// TIA Portal project "Event Logger Example" (V15.1)

(* hardware
DEVICE "S71500/ET200MP station_1"  S7-1500 station
   slot 0: "Rail_0"  Rack  6ES7 590-1***0-0AA0
   slot 1: "Event Example"  CPU 1511-1 PN  6ES7 511-1AK00-0AB0  V1.8
      slot 3: "CPU display_1"  6ES7591-1AA00-0AA0
*)

// ===== PLC "Event Example"  CPU 1511-1 PN =====

VAR_GLOBAL   // PLC tag table "Default tag table"
   "System_Byte" AT %MB1 : Byte;
   "FirstScan" AT %M1.0 : Bool;
   "DiagStatusUpdate" AT %M1.1 : Bool;
   "AlwaysTRUE" AT %M1.2 : Bool;
   "AlwaysFALSE" AT %M1.3 : Bool;
   "Clock_Byte" AT %MB0 : Byte;
   "Clock_10Hz" AT %M0.0 : Bool;
   "Clock_5Hz" AT %M0.1 : Bool;
   "Clock_2.5Hz" AT %M0.2 : Bool;
   "Clock_2Hz" AT %M0.3 : Bool;
   "Clock_1.25Hz" AT %M0.4 : Bool;
   "Clock_1Hz" AT %M0.5 : Bool;
   "Clock_0.625Hz" AT %M0.6 : Bool;
   "Clock_0.5Hz" AT %M0.7 : Bool;
   "mSendKeepAlive" AT %M2.0 : Bool;
END_VAR

TYPE "EventDataToPC"
   STRUCT
      EventCode : DInt;
      Par1 : DInt;
      Par2 : DInt;
      Par3 : DInt;
      Par4 : DInt;
      Par5 : DInt;
      Par6 : DInt;
      Par7 : DInt;
      Par8 : DInt;
   END_STRUCT;
END_TYPE

TYPE "KeepAliveToPC"
   STRUCT
      MessageType : DInt := 12;
      Flags : DInt := 1;
   END_STRUCT;
END_TYPE

DATA_BLOCK "event_IDB"   // DB12
{ S7_Optimized_Access := 'TRUE' }
VERSION : 0.1
// stored: InstanceOfName ET_GeneralEventToBuffer
"ET_GeneralEventToBuffer"
BEGIN
END_DATA_BLOCK

// folder: System blocks/Program resources

DATA_BLOCK "PCComms_ConnectDly"   // DB1
{ S7_Optimized_Access := 'TRUE' }
AUTHOR : Simatic
FAMILY : IEC
NAME : IEC_TMR
VERSION : 1.0
// stored: InstanceOfName IEC_TIMER
"IEC_TIMER"
BEGIN
END_DATA_BLOCK

DATA_BLOCK "PCComms_SendRequestTimeout"   // DB6
{ S7_Optimized_Access := 'TRUE' }
AUTHOR : Simatic
FAMILY : IEC
NAME : IEC_TMR
VERSION : 1.0
// stored: InstanceOfName IEC_TIMER
"IEC_TIMER"
BEGIN
END_DATA_BLOCK

DATA_BLOCK "tKeepAlive"   // DB8
{ S7_Optimized_Access := 'TRUE' }
AUTHOR : Simatic
FAMILY : IEC
NAME : IEC_TMR
VERSION : 1.0
// stored: InstanceOfName IEC_TIMER
"IEC_TIMER"
BEGIN
END_DATA_BLOCK

DATA_BLOCK "PCComms_DisconnectDly"   // DB9
{ S7_Optimized_Access := 'TRUE' }
AUTHOR : Simatic
FAMILY : IEC
NAME : IEC_TMR
VERSION : 1.0
// stored: InstanceOfName IEC_TIMER
"IEC_TIMER"
BEGIN
END_DATA_BLOCK

DATA_BLOCK "PCComms_ReconnectDly"   // DB11
{ S7_Optimized_Access := 'TRUE' }
AUTHOR : Simatic
FAMILY : IEC
NAME : IEC_TMR
VERSION : 1.0
// stored: InstanceOfName IEC_TIMER
"IEC_TIMER"
BEGIN
END_DATA_BLOCK

DATA_BLOCK "tEventCycler"   // DB13
{ S7_Optimized_Access := 'TRUE' }
AUTHOR : Simatic
FAMILY : IEC
NAME : IEC_TMR
VERSION : 1.0
// stored: InstanceOfName IEC_TIMER
"IEC_TIMER"
BEGIN
END_DATA_BLOCK

// folder: _EventTracking

DATA_BLOCK "PCComms_Data"   // DB300
{ S7_Optimized_Access := 'FALSE' }
VERSION : 0.1
   VAR
      CON : Struct
         RequestConnection : Bool;
         RequestReconnection : Bool;
         ErrorStatus : Word;
         ManualConnect : Bool;
         ConnectRequestONS : Bool;
         ReconnectRequestONS : Bool;
         KeepAliveONS : Bool;
      END_STRUCT;
      DIAG : Struct
         ErrorStatus : Word;
         Request : Bool;
         Result : TDiag_Status;
         NumberOfSuccesses : Int := 0;
         State : Struct
            NoConnectionData : Bool;
            ConnectionTerminated : Bool;
            EstablishingConnection : Bool;
            WaitingForConnection : Bool;
            ConnectionEstablished : Bool;
            ConnectionBeingTerminated : Bool;
            UnknownState : Bool;
            HMIState : Int;
         END_STRUCT;
      END_STRUCT;
      DISCON : Struct
         ErrorStatus : Word;
         DisconnectRequest : Bool;
         ReconnectRequest : Bool;
      END_STRUCT;
      TX : Struct
         NumberOfSuccesfulSends : Int;
         HeadPointer : Int;
         TailPointer : Int;
         MaxPointer : Int := 9;
         SendRequest : Bool;
         ManualTestWithDummyData : Bool;
         DataLengthIn : UDInt;
         DataIn : Struct
            DataLength : DInt;
            Data : Array[0..1023] of Byte;
         END_STRUCT;
         DataOut : Struct
            DataLength : DInt;
            Data : Array[0..1023] of Byte;
         END_STRUCT;
         DataBuffer : Array[0..9] of Struct
            DataLength : DInt;
            Data : Array[0..1023] of Byte;
         END_STRUCT;
         StatusSaved : Word;
      END_STRUCT;
      RX : Struct
         BytesReceived : Int;
         StatusSaved : Word;
         Data : Array[0..254] of Byte;
         NumberOfSuccesfulReceives : Int;
      END_STRUCT;
      EventDataToPC : "EventDataToPC";
      KeepAliveToPC : "KeepAliveToPC";
      Alarms : Array[0..31] of Bool;
   END_VAR
BEGIN
   Alarms[0] := FALSE;
   Alarms[1] := FALSE;
   Alarms[2] := FALSE;
   Alarms[3] := FALSE;
   Alarms[4] := FALSE;
   Alarms[5] := FALSE;
   Alarms[6] := FALSE;
   Alarms[7] := FALSE;
   Alarms[8] := FALSE;
   Alarms[9] := FALSE;
   Alarms[10] := FALSE;
   Alarms[11] := FALSE;
   Alarms[12] := FALSE;
   Alarms[13] := FALSE;
   Alarms[14] := FALSE;
   Alarms[15] := FALSE;
   Alarms[16] := FALSE;
   Alarms[17] := FALSE;
   Alarms[18] := FALSE;
   Alarms[19] := FALSE;
   Alarms[20] := FALSE;
   Alarms[21] := FALSE;
   Alarms[22] := FALSE;
   Alarms[23] := FALSE;
   Alarms[24] := FALSE;
   Alarms[25] := FALSE;
   Alarms[26] := FALSE;
   Alarms[27] := FALSE;
   Alarms[28] := FALSE;
   Alarms[29] := FALSE;
   Alarms[30] := FALSE;
   Alarms[31] := FALSE;
END_DATA_BLOCK

DATA_BLOCK "ET_TxBuffer"   // DB306
{ S7_Optimized_Access := 'TRUE' }
VERSION : 0.1
   VAR
      NextAddPoint : Int;
      LastSendPoint : Int;
      SendEvtDataToPCReq : Bool;
      Buffer : Array[1..10] of "EventDataToPC";
   END_VAR
BEGIN
END_DATA_BLOCK

DATA_BLOCK "ET_Alarms"   // DB552
{ S7_Optimized_Access := 'FALSE' }
VERSION : 0.1
   VAR
      EventCommsFlt : Bool;
   END_VAR
BEGIN
END_DATA_BLOCK

DATA_BLOCK "PCComms_Connection_DB"   // DB555
{ S7_Optimized_Access := 'TRUE' }
AUTHOR : SIMATIC
FAMILY : MC7Plus
NAME : TC_IP_v4
VERSION : 1.0
// stored: InstanceOfName TCON_IP_v4
"TCON_IP_v4"
BEGIN
   ID := 2;
   InterfaceId := 64;
   LocalPort := 2000;
   RemotePort := 10200;
   RemoteAddress.ADDR[1] := 192;
   RemoteAddress.ADDR[2] := 168;
   RemoteAddress.ADDR[3] := 100;
   RemoteAddress.ADDR[4] := 253;
END_DATA_BLOCK

DATA_BLOCK "ET_GeneralData"   // DB700
{ S7_Optimized_Access := 'TRUE' }
VERSION : 0.1
   VAR RETAIN
      LogTrackingDiagEnabled : Bool := TRUE;   // True = Log Tracking Diagnostics Code Is Enabled. Diag Data Will Be Sent To PC
   END_VAR
   VAR
      NewDataReceived : Bool;   // True = New Log Data Was Received (New Memory Number) From Cant Saw
      UpdatedDataReceived : Bool;   // True = Updated Data Was Received (Same Memory Number) From Cant Saw
      LogLoadingToLine : Bool;   // True = Log Being Loaded To The Line
      MemoryToRemove : Int;   // Memory Number To Remove From The Line
      LastMemoryReceived : Int;   // Last Memory Number Received From Cant Saw CPU
      ReconnectTrigger : Bool;
      ReconnectPulseONS : Bool;
      TSendDone : Bool;
      TSendError : Bool;
      ErrorTrap_TCON : Bool;
   END_VAR
BEGIN
END_DATA_BLOCK

DATA_BLOCK "ET_EventDataTxBuffer"   // DB740
{ S7_Optimized_Access := 'TRUE' }
VERSION : 0.1
   VAR
      NextAddPoint : Int;   // Pointer To The Next Place To Add Data To The Buffer
      LastSendPoint : Int;   // Pointer To The Last Data That Was Sent
      SendDataToPCReq : Bool;
      ErrorTrapTSEND : Word;
      ErrorTrapTCON : Word;
      Buffer : Array[1..10] of Struct   // Buffer Of Data To Be Sent To The Scanner Applications
         Data : Array[0..31] of Int;   // Data To Be Sent (Has No Struct As Items Change Depending On Packet Type)
      END_STRUCT;
   END_VAR
BEGIN
END_DATA_BLOCK

// folder: (top level)

ORGANIZATION_BLOCK "Main"   // OB1, LAD, ProgramCycle
TITLE = "Main Program Sweep (Cycle)"
{ S7_Optimized_Access := 'TRUE' }
VERSION : 0.1
   VAR_INPUT
      Initial_Call : Bool;   // Initial call of this OB
      Remanence : Bool;   // =True, if remanent data are available
   END_VAR
BEGIN

REGION Network 1 (STL): Call the comms functions
         CALL  "PCComms_Communications";
END_REGION

REGION Network 2: Send an event every 30 seconds.
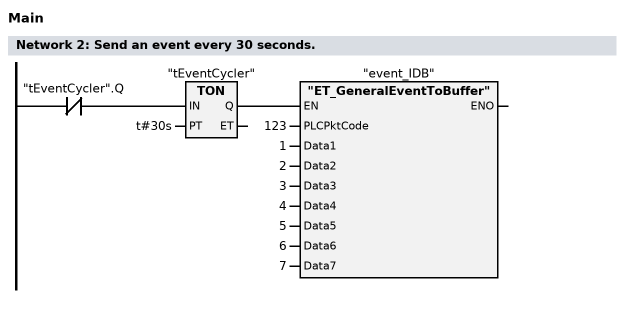
   "tEventCycler".TON(IN := NOT "tEventCycler".Q, PT := t#30s);
   IF "tEventCycler".Q THEN
       "event_IDB"(PLCPktCode := 123,   // "ET_GeneralEventToBuffer"
                   Data1 := 1,
                   Data2 := 2,
                   Data3 := 3,
                   Data4 := 4,
                   Data5 := 5,
                   Data6 := 6,
                   Data7 := 7);
   END_IF;
END_REGION
END_ORGANIZATION_BLOCK

// folder: _EventTracking

FUNCTION_BLOCK "ET_GeneralEventToBuffer"   // FB34, SCL
{ S7_Optimized_Access := 'TRUE' }
VERSION : 0.1
   VAR_INPUT
      PLCPktCode : Int := 80;
      Data1 : Int;
      Data2 : Int;
      Data3 : Int;
      Data4 : Int;
      Data5 : Int;
      Data6 : Int;
      Data7 : Int;
   END_VAR
   VAR_TEMP
      i : Int;
      OneShoot : Bool;
      AddPoint : Int;   // Pointer to the point to add data to in the buffer
      BoardCount : Int;
   END_VAR
   VAR CONSTANT
      SOPCode : Int := -1;
      EOPCode : Int := -99;
      DataPktLength : Int := 64;
   END_VAR
BEGIN

   // Increment write pointer
   "ET_TxBuffer".NextAddPoint := "ET_TxBuffer".NextAddPoint + 1;
   IF "ET_TxBuffer".NextAddPoint > 10 THEN
       "ET_TxBuffer".NextAddPoint := 1;
   END_IF;
   #AddPoint := "ET_TxBuffer".NextAddPoint;

   // Write data into buffer at write point
   "ET_TxBuffer".Buffer[#AddPoint].EventCode := 50;//#EventCode;
   "ET_TxBuffer".Buffer[#AddPoint].Par1 := #PLCPktCode;
   "ET_TxBuffer".Buffer[#AddPoint].Par2 := #Data1;
   "ET_TxBuffer".Buffer[#AddPoint].Par3 := #Data2;
   "ET_TxBuffer".Buffer[#AddPoint].Par4 := #Data3;
   "ET_TxBuffer".Buffer[#AddPoint].Par5 := #Data4;
   "ET_TxBuffer".Buffer[#AddPoint].Par6 := #Data5;
   "ET_TxBuffer".Buffer[#AddPoint].Par7 := #Data6;
   "ET_TxBuffer".Buffer[#AddPoint].Par8 := #Data7;

   ENO := true;
END_FUNCTION_BLOCK

FUNCTION "PCComms_Reconection" : Void   // FC90, LAD
TITLE = Reconnection Routine - only use if PLC is active end
{ S7_Optimized_Access := 'TRUE' }
VERSION : 0.1
// We suspect that the disconnection/reconnection is only necessary if the PLC is the active end.  If the PLC is the passive (server) end then it can just sit listening all day without having to disconnect/reconnect.
   VAR_TEMP   // added for the SCL form of the ladder/FBD networks
      _w1 : Bool;
   END_VAR
BEGIN

REGION Network 1: Force a Disconnection if there has been no connection made in 20s
   // We suspect that the disconnection/reconnection is only necessary if the PLC is the active end.  If the PLC is the passive (server) end then it can just sit listening all day without having to disconnect/reconnect.
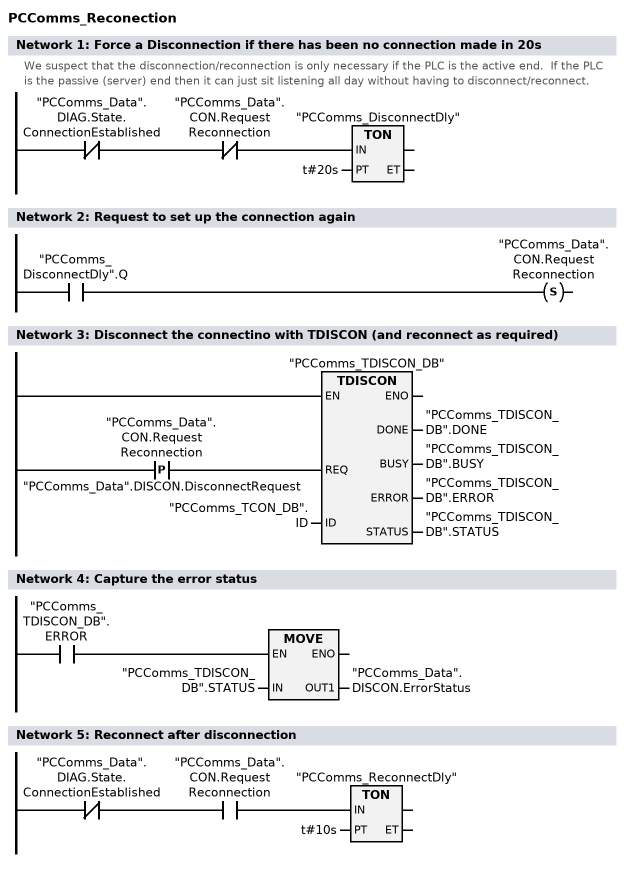
   "PCComms_DisconnectDly".TON(IN := NOT "PCComms_Data".DIAG.State.ConnectionEstablished AND NOT "PCComms_Data".CON.RequestReconnection,
                           PT := t#20s);
END_REGION

REGION Network 2: Request to set up the connection again
   RUNG wire#powerrail
      Contact( "PCComms_DisconnectDly".Q )
      S_Coil( "PCComms_Data".CON.RequestReconnection )
   END_RUNG
   // the same network as SCL:
   IF "PCComms_DisconnectDly".Q THEN "PCComms_Data".CON.RequestReconnection := TRUE; END_IF;
END_REGION

REGION Network 3: Disconnect the connectino with TDISCON (and reconnect as required)
   #_w1 := "PCComms_Data".CON.RequestReconnection AND NOT "PCComms_Data".DISCON.DisconnectRequest;   // rising edge of "PCComms_Data".CON.RequestReconnection
   "PCComms_Data".DISCON.DisconnectRequest := "PCComms_Data".CON.RequestReconnection;
   "PCComms_TDISCON_DB"(REQ := #_w1,   // TDISCON
                        ID := "PCComms_TCON_DB".ID,
                        DONE => "PCComms_TDISCON_DB".DONE,
                        BUSY => "PCComms_TDISCON_DB".BUSY,
                        ERROR => "PCComms_TDISCON_DB".ERROR,
                        STATUS => "PCComms_TDISCON_DB".STATUS);
END_REGION

REGION Network 4: Capture the error status
   RUNG wire#powerrail
      Contact( "PCComms_TDISCON_DB".ERROR )
      Move(in := "PCComms_TDISCON_DB".STATUS, out1 => "PCComms_Data".DISCON.ErrorStatus)
   END_RUNG
   // the same network as SCL:
   IF "PCComms_TDISCON_DB".ERROR THEN
       "PCComms_Data".DISCON.ErrorStatus := "PCComms_TDISCON_DB".STATUS;
   END_IF;
END_REGION

REGION Network 5: Reconnect after disconnection
   "PCComms_ReconnectDly".TON(IN := NOT "PCComms_Data".DIAG.State.ConnectionEstablished AND "PCComms_Data".CON.RequestReconnection,
                           PT := t#10s);
END_REGION
END_FUNCTION

FUNCTION "PCComms_ProcessTxMessages" : Void   // FC91, LAD
TITLE = Manage the connection and data transmit and receive.
{ S7_Optimized_Access := 'TRUE' }
VERSION : 0.1
   VAR_TEMP
      RETVAL : DInt;
      BufferPos : DInt;   // Pos for the serialize function
   END_VAR
   VAR_TEMP   // added for the SCL form of the ladder/FBD networks
      _w1 : Bool;
      _w2 : Bool;
   END_VAR
BEGIN

REGION Network 1: If no comms packets sent, send a keep alive.
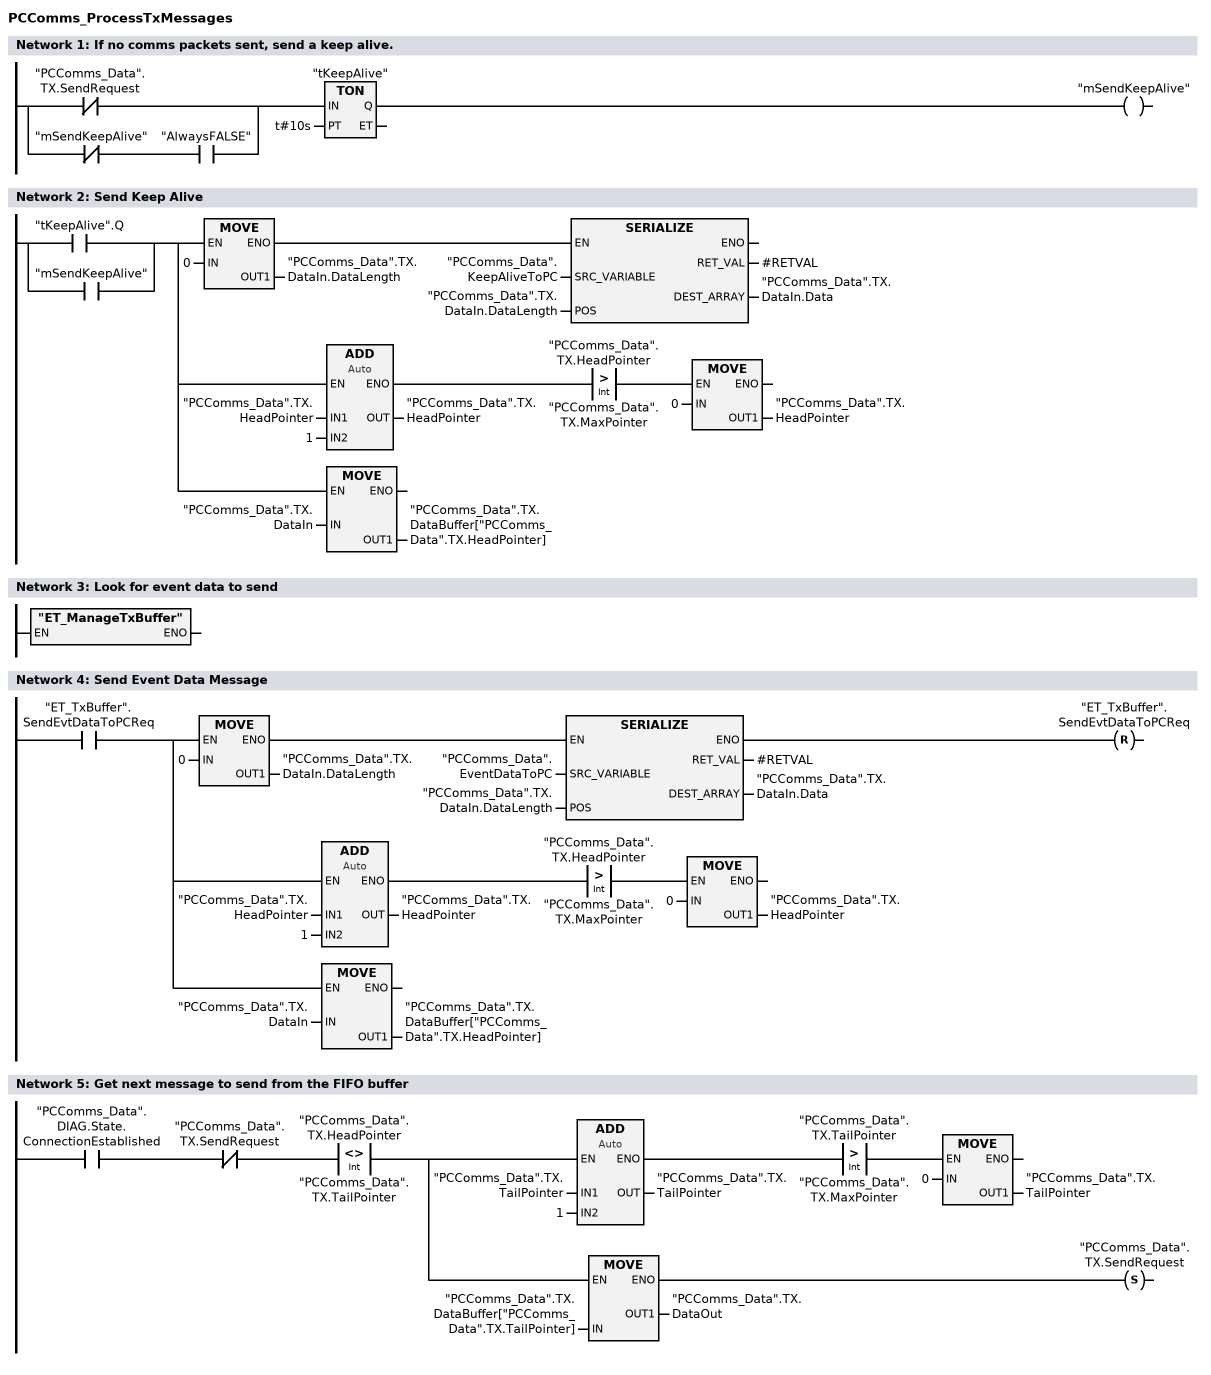
   "tKeepAlive".TON(IN := NOT "PCComms_Data".TX.SendRequest OR (NOT "mSendKeepAlive" AND "AlwaysFALSE"),
                    PT := t#10s);
   "mSendKeepAlive" := "tKeepAlive".Q;
END_REGION

REGION Network 2: Send Keep Alive
   // no SCL statement known for Serialize: written as a call
   #_w1 := "tKeepAlive".Q OR "mSendKeepAlive";
   IF #_w1 THEN
       "PCComms_Data".TX.DataIn.DataLength := 0;
       #RETVAL := Serialize(SRC_VARIABLE := "PCComms_Data".KeepAliveToPC,
                            POS := "PCComms_Data".TX.DataIn.DataLength,
                            DEST_ARRAY => "PCComms_Data".TX.DataIn.Data);
       "PCComms_Data".TX.HeadPointer := "PCComms_Data".TX.HeadPointer + 1;
   END_IF;
   IF #_w1 AND ("PCComms_Data".TX.HeadPointer > "PCComms_Data".TX.MaxPointer) THEN
       "PCComms_Data".TX.HeadPointer := 0;
   END_IF;
   IF #_w1 THEN
       "PCComms_Data".TX.DataBuffer["PCComms_Data".TX.HeadPointer] := "PCComms_Data".TX.DataIn;
   END_IF;
END_REGION

REGION Network 3: Look for event data to send
   RUNG wire#powerrail
      "ET_ManageTxBuffer"()
   END_RUNG
   // the same network as SCL:
   "ET_ManageTxBuffer"();
END_REGION

REGION Network 4: Send Event Data Message
   // no SCL statement known for Serialize: written as a call
   // ENO of a box is taken as its EN; it also drops when the box reports an error
   IF "ET_TxBuffer".SendEvtDataToPCReq THEN "PCComms_Data".TX.DataIn.DataLength := 0; END_IF;
   #_w1 := "ET_TxBuffer".SendEvtDataToPCReq;
   #_w2 := "ET_TxBuffer".SendEvtDataToPCReq;
   IF #_w2 THEN
       #RETVAL := Serialize(SRC_VARIABLE := "PCComms_Data".EventDataToPC,
                            POS := "PCComms_Data".TX.DataIn.DataLength,
                            DEST_ARRAY => "PCComms_Data".TX.DataIn.Data);
       "ET_TxBuffer".SendEvtDataToPCReq := FALSE;
   END_IF;
   IF #_w1 THEN "PCComms_Data".TX.HeadPointer := "PCComms_Data".TX.HeadPointer + 1; END_IF;
   IF #_w1 AND ("PCComms_Data".TX.HeadPointer > "PCComms_Data".TX.MaxPointer) THEN
       "PCComms_Data".TX.HeadPointer := 0;
   END_IF;
   IF #_w1 THEN
       "PCComms_Data".TX.DataBuffer["PCComms_Data".TX.HeadPointer] := "PCComms_Data".TX.DataIn;
   END_IF;
END_REGION

REGION Network 5: Get next message to send from the FIFO buffer
   RUNG wire#powerrail
      Contact( "PCComms_Data".DIAG.State.ConnectionEstablished )
      I_Contact( "PCComms_Data".TX.SendRequest )
      { S7_Templates := "SrcType := Int" } NE_Contact(in1 := "PCComms_Data".TX.HeadPointer, in2 := "PCComms_Data".TX.TailPointer)
      wire#w1
      Add(in1 := "PCComms_Data".TX.TailPointer, in2 := 1, out => "PCComms_Data".TX.TailPointer)
      { S7_Templates := "SrcType := Int" } GT_Contact(in1 := "PCComms_Data".TX.TailPointer, in2 := "PCComms_Data".TX.MaxPointer)
      Move(in := 0, out1 => "PCComms_Data".TX.TailPointer)
   END_RUNG
   RUNG wire#w1
      Move(in := "PCComms_Data".TX.DataBuffer["PCComms_Data".TX.TailPointer], out1 => "PCComms_Data".TX.DataOut)
      S_Coil( "PCComms_Data".TX.SendRequest )
   END_RUNG
   // the same network as SCL:
   #_w1 := "PCComms_Data".DIAG.State.ConnectionEstablished AND NOT "PCComms_Data".TX.SendRequest AND ("PCComms_Data".TX.HeadPointer <> "PCComms_Data".TX.TailPointer);
   IF #_w1 THEN "PCComms_Data".TX.TailPointer := "PCComms_Data".TX.TailPointer + 1; END_IF;
   IF #_w1 AND ("PCComms_Data".TX.TailPointer > "PCComms_Data".TX.MaxPointer) THEN
       "PCComms_Data".TX.TailPointer := 0;
   END_IF;
   IF #_w1 THEN
       "PCComms_Data".TX.DataOut := "PCComms_Data".TX.DataBuffer["PCComms_Data".TX.TailPointer];
       "PCComms_Data".TX.SendRequest := TRUE;
   END_IF;
END_REGION
END_FUNCTION

FUNCTION "PCComms_Communications" : Void   // FC740, LAD
TITLE = Event Tracking Comms Management
{ S7_Optimized_Access := 'TRUE' }
VERSION : 0.1
   VAR_TEMP
      AG_SEND_Done : Bool;   // AG_SEND Has Been Done
      AG_SEND_Error : Bool;   // AG_SEND Has An Error
      AG_SEND_Status : Word;   // AG_SEND Status
      DISCON_Done : Bool;
   END_VAR
   VAR CONSTANT
      TCON_ID : Conn_Ouc := 16#0091;
   END_VAR
   VAR_TEMP   // added for the SCL form of the ladder/FBD networks
      _w1 : Bool;
      _w2 : Bool;
      _w3 : Bool;
   END_VAR
BEGIN

REGION Network 1: Delay starting the comms until the PLC starts up.
   // Not sure if this is really necessary.
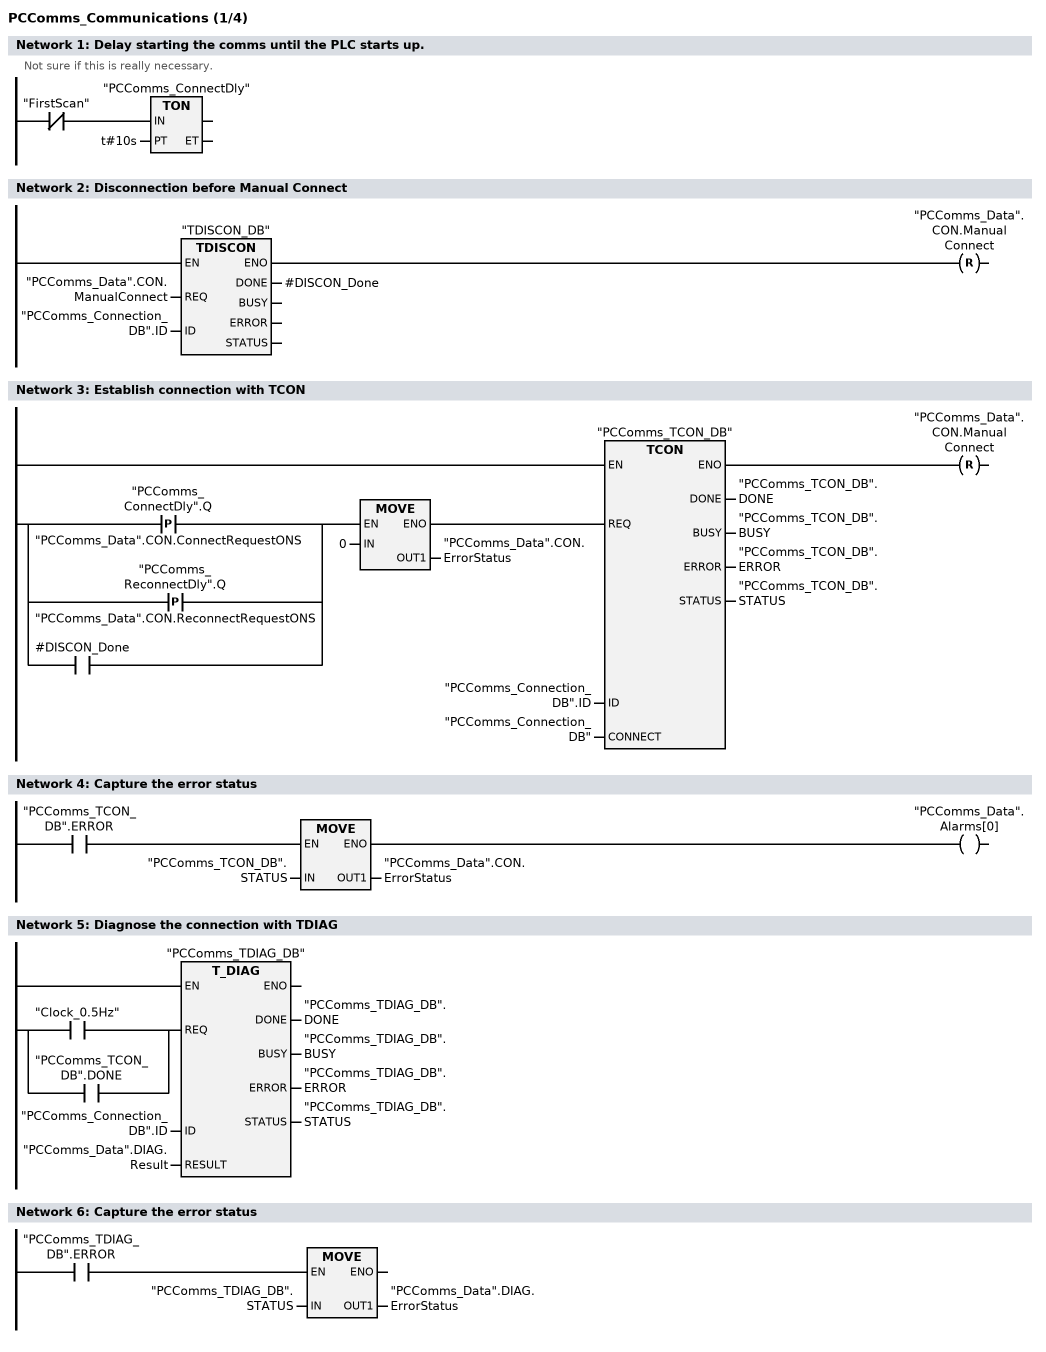
   "PCComms_ConnectDly".TON(IN := NOT "FirstScan", PT := t#10s);
END_REGION

REGION Network 2: Disconnection before Manual Connect
   // ENO of a box is taken as its EN; it also drops when the box reports an error
   "TDISCON_DB"(REQ := "PCComms_Data".CON.ManualConnect, ID := "PCComms_Connection_DB".ID, DONE => #DISCON_Done);   // TDISCON
   "PCComms_Data".CON.ManualConnect := FALSE;
END_REGION

REGION Network 3: Establish connection with TCON
   // ENO of a box is taken as its EN; it also drops when the box reports an error
   #_w1 := "PCComms_ConnectDly".Q AND NOT "PCComms_Data".CON.ConnectRequestONS;   // rising edge of "PCComms_ConnectDly".Q
   "PCComms_Data".CON.ConnectRequestONS := "PCComms_ConnectDly".Q;
   #_w2 := "PCComms_ReconnectDly".Q AND NOT "PCComms_Data".CON.ReconnectRequestONS;   // rising edge of "PCComms_ReconnectDly".Q
   "PCComms_Data".CON.ReconnectRequestONS := "PCComms_ReconnectDly".Q;
   #_w3 := #_w1 OR #_w2 OR #DISCON_Done;
   IF #_w3 THEN "PCComms_Data".CON.ErrorStatus := 0; END_IF;
   "PCComms_TCON_DB"(REQ := #_w3,   // TCON
                     ID := "PCComms_Connection_DB".ID,
                     CONNECT := "PCComms_Connection_DB",
                     DONE => "PCComms_TCON_DB".DONE,
                     BUSY => "PCComms_TCON_DB".BUSY,
                     ERROR => "PCComms_TCON_DB".ERROR,
                     STATUS => "PCComms_TCON_DB".STATUS);
   "PCComms_Data".CON.ManualConnect := FALSE;
END_REGION

REGION Network 4: Capture the error status
   RUNG wire#powerrail
      Contact( "PCComms_TCON_DB".ERROR )
      Move(in := "PCComms_TCON_DB".STATUS, out1 => "PCComms_Data".CON.ErrorStatus)
      Coil( "PCComms_Data".Alarms[0] )
   END_RUNG
   // the same network as SCL:
   IF "PCComms_TCON_DB".ERROR THEN "PCComms_Data".CON.ErrorStatus := "PCComms_TCON_DB".STATUS; END_IF;
   "PCComms_Data".Alarms[0] := "PCComms_TCON_DB".ERROR;
END_REGION

REGION Network 5: Diagnose the connection with TDIAG
   "PCComms_TDIAG_DB"(REQ := "Clock_0.5Hz" OR "PCComms_TCON_DB".DONE,   // T_DIAG
                      ID := "PCComms_Connection_DB".ID,
                      RESULT := "PCComms_Data".DIAG.Result,
                      DONE => "PCComms_TDIAG_DB".DONE,
                      BUSY => "PCComms_TDIAG_DB".BUSY,
                      ERROR => "PCComms_TDIAG_DB".ERROR,
                      STATUS => "PCComms_TDIAG_DB".STATUS);
END_REGION

REGION Network 6: Capture the error status
   RUNG wire#powerrail
      Contact( "PCComms_TDIAG_DB".ERROR )
      Move(in := "PCComms_TDIAG_DB".STATUS, out1 => "PCComms_Data".DIAG.ErrorStatus)
   END_RUNG
   // the same network as SCL:
   IF "PCComms_TDIAG_DB".ERROR THEN "PCComms_Data".DIAG.ErrorStatus := "PCComms_TDIAG_DB".STATUS; END_IF;
END_REGION

REGION Network 7: Interpret the connection status
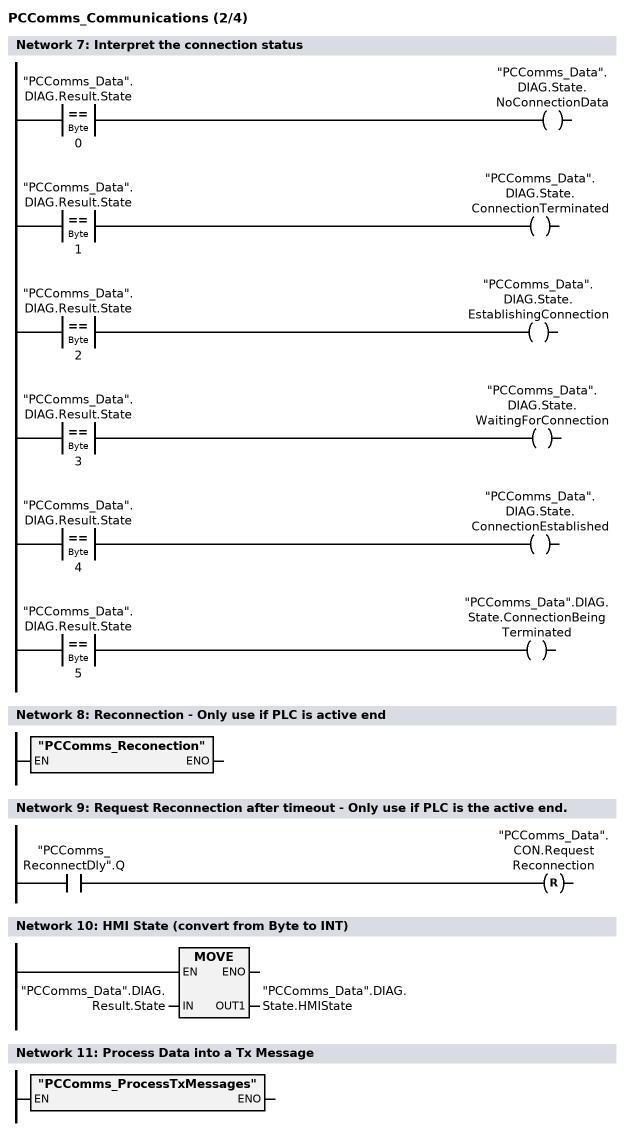
   RUNG wire#powerrail
      { S7_Templates := "SrcType := Byte" } EQ_Contact(in1 := "PCComms_Data".DIAG.Result.State, in2 := 0)
      Coil( "PCComms_Data".DIAG.State.NoConnectionData )
   END_RUNG
   RUNG wire#powerrail
      { S7_Templates := "SrcType := Byte" } EQ_Contact(in1 := "PCComms_Data".DIAG.Result.State, in2 := 1)
      Coil( "PCComms_Data".DIAG.State.ConnectionTerminated )
   END_RUNG
   RUNG wire#powerrail
      { S7_Templates := "SrcType := Byte" } EQ_Contact(in1 := "PCComms_Data".DIAG.Result.State, in2 := 2)
      Coil( "PCComms_Data".DIAG.State.EstablishingConnection )
   END_RUNG
   RUNG wire#powerrail
      { S7_Templates := "SrcType := Byte" } EQ_Contact(in1 := "PCComms_Data".DIAG.Result.State, in2 := 3)
      Coil( "PCComms_Data".DIAG.State.WaitingForConnection )
   END_RUNG
   RUNG wire#powerrail
      { S7_Templates := "SrcType := Byte" } EQ_Contact(in1 := "PCComms_Data".DIAG.Result.State, in2 := 4)
      Coil( "PCComms_Data".DIAG.State.ConnectionEstablished )
   END_RUNG
   RUNG wire#powerrail
      { S7_Templates := "SrcType := Byte" } EQ_Contact(in1 := "PCComms_Data".DIAG.Result.State, in2 := 5)
      Coil( "PCComms_Data".DIAG.State.ConnectionBeingTerminated )
   END_RUNG
   // the same network as SCL:
   "PCComms_Data".DIAG.State.NoConnectionData := "PCComms_Data".DIAG.Result.State = 0;
   "PCComms_Data".DIAG.State.ConnectionTerminated := "PCComms_Data".DIAG.Result.State = 1;
   "PCComms_Data".DIAG.State.EstablishingConnection := "PCComms_Data".DIAG.Result.State = 2;
   "PCComms_Data".DIAG.State.WaitingForConnection := "PCComms_Data".DIAG.Result.State = 3;
   "PCComms_Data".DIAG.State.ConnectionEstablished := "PCComms_Data".DIAG.Result.State = 4;
   "PCComms_Data".DIAG.State.ConnectionBeingTerminated := "PCComms_Data".DIAG.Result.State = 5;
END_REGION

REGION Network 8: Reconnection - Only use if PLC is active end
   RUNG wire#powerrail
      "PCComms_Reconection"()
   END_RUNG
   // the same network as SCL:
   "PCComms_Reconection"();
END_REGION

REGION Network 9: Request Reconnection after timeout - Only use if PLC is the active end.
   RUNG wire#powerrail
      Contact( "PCComms_ReconnectDly".Q )
      R_Coil( "PCComms_Data".CON.RequestReconnection )
   END_RUNG
   // the same network as SCL:
   IF "PCComms_ReconnectDly".Q THEN "PCComms_Data".CON.RequestReconnection := FALSE; END_IF;
END_REGION

REGION Network 10: HMI State (convert from Byte to INT)
   RUNG wire#powerrail
      Move(in := "PCComms_Data".DIAG.Result.State, out1 => "PCComms_Data".DIAG.State.HMIState)
   END_RUNG
   // the same network as SCL:
   "PCComms_Data".DIAG.State.HMIState := "PCComms_Data".DIAG.Result.State;
END_REGION

REGION Network 11: Process Data into a Tx Message
   RUNG wire#powerrail
      "PCComms_ProcessTxMessages"()
   END_RUNG
   // the same network as SCL:
   "PCComms_ProcessTxMessages"();
END_REGION

REGION Network 12: Send Data with TSEND
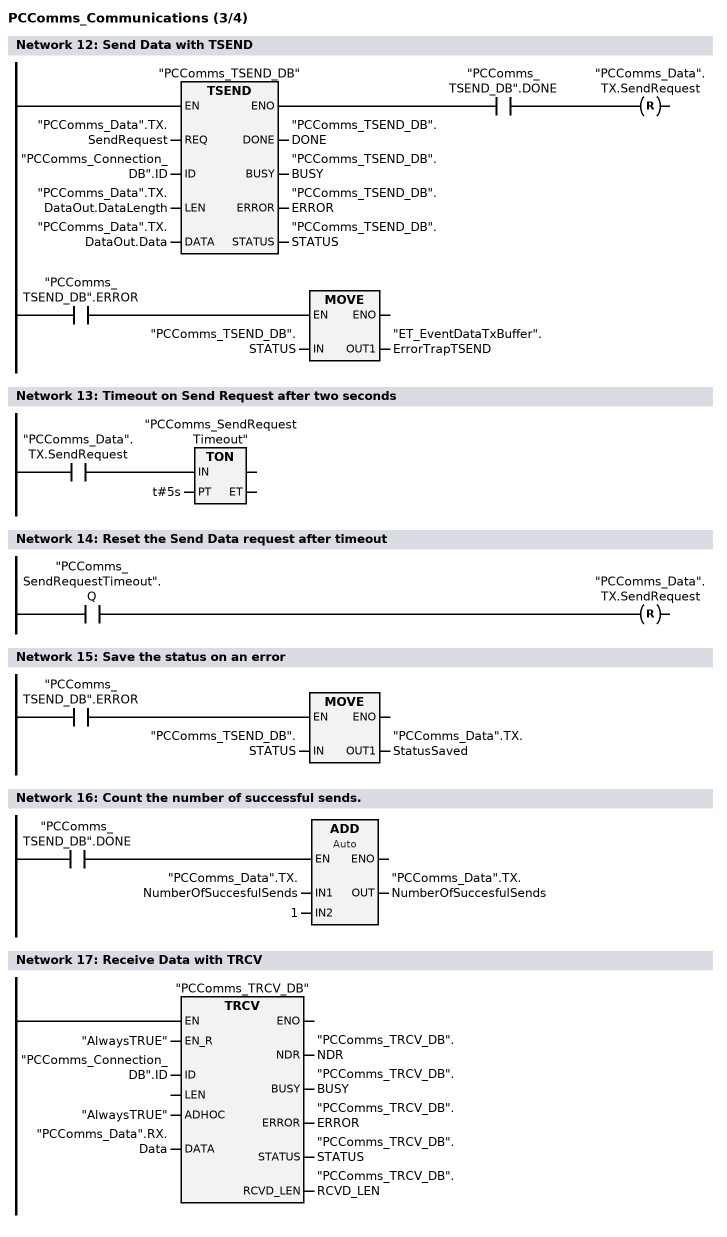
   // ENO of a box is taken as its EN; it also drops when the box reports an error
   "PCComms_TSEND_DB"(REQ := "PCComms_Data".TX.SendRequest,   // TSEND
                      ID := "PCComms_Connection_DB".ID,
                      LEN := "PCComms_Data".TX.DataOut.DataLength,
                      DATA := "PCComms_Data".TX.DataOut.Data,
                      DONE => "PCComms_TSEND_DB".DONE,
                      BUSY => "PCComms_TSEND_DB".BUSY,
                      ERROR => "PCComms_TSEND_DB".ERROR,
                      STATUS => "PCComms_TSEND_DB".STATUS);
   IF "PCComms_TSEND_DB".DONE THEN "PCComms_Data".TX.SendRequest := FALSE; END_IF;
   IF "PCComms_TSEND_DB".ERROR THEN
       "ET_EventDataTxBuffer".ErrorTrapTSEND := "PCComms_TSEND_DB".STATUS;
   END_IF;
END_REGION

REGION Network 13: Timeout on Send Request after two seconds
   "PCComms_SendRequestTimeout".TON(IN := "PCComms_Data".TX.SendRequest, PT := t#5s);
END_REGION

REGION Network 14: Reset the Send Data request after timeout
   RUNG wire#powerrail
      Contact( "PCComms_SendRequestTimeout".Q )
      R_Coil( "PCComms_Data".TX.SendRequest )
   END_RUNG
   // the same network as SCL:
   IF "PCComms_SendRequestTimeout".Q THEN "PCComms_Data".TX.SendRequest := FALSE; END_IF;
END_REGION

REGION Network 15: Save the status on an error
   RUNG wire#powerrail
      Contact( "PCComms_TSEND_DB".ERROR )
      Move(in := "PCComms_TSEND_DB".STATUS, out1 => "PCComms_Data".TX.StatusSaved)
   END_RUNG
   // the same network as SCL:
   IF "PCComms_TSEND_DB".ERROR THEN "PCComms_Data".TX.StatusSaved := "PCComms_TSEND_DB".STATUS; END_IF;
END_REGION

REGION Network 16: Count the number of successful sends.
   RUNG wire#powerrail
      Contact( "PCComms_TSEND_DB".DONE )
      Add(in1 := "PCComms_Data".TX.NumberOfSuccesfulSends, in2 := 1, out => "PCComms_Data".TX.NumberOfSuccesfulSends)
   END_RUNG
   // the same network as SCL:
   IF "PCComms_TSEND_DB".DONE THEN
       "PCComms_Data".TX.NumberOfSuccesfulSends := "PCComms_Data".TX.NumberOfSuccesfulSends + 1;
   END_IF;
END_REGION

REGION Network 17: Receive Data with TRCV
   "PCComms_TRCV_DB"(EN_R := "AlwaysTRUE",   // TRCV
                     ID := "PCComms_Connection_DB".ID,
                     ADHOC := "AlwaysTRUE",
                     DATA := "PCComms_Data".RX.Data,
                     NDR => "PCComms_TRCV_DB".NDR,
                     BUSY => "PCComms_TRCV_DB".BUSY,
                     ERROR => "PCComms_TRCV_DB".ERROR,
                     STATUS => "PCComms_TRCV_DB".STATUS,
                     RCVD_LEN => "PCComms_TRCV_DB".RCVD_LEN);
END_REGION

REGION Network 18: Copy the length of data received and count the number of succesful receives.
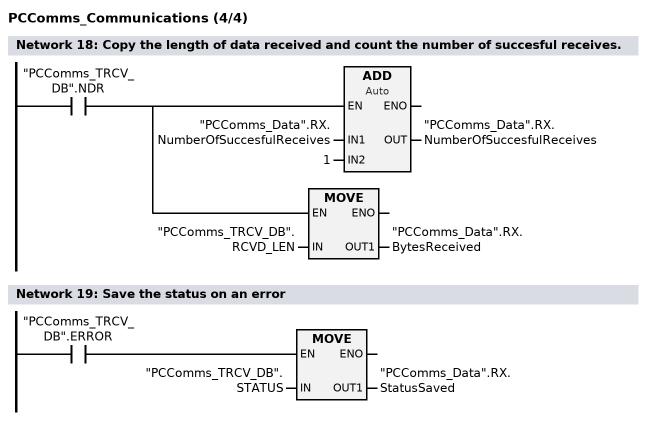
   RUNG wire#powerrail
      Contact( "PCComms_TRCV_DB".NDR )
      wire#w1
      Add(in1 := "PCComms_Data".RX.NumberOfSuccesfulReceives, in2 := 1, out => "PCComms_Data".RX.NumberOfSuccesfulReceives)
   END_RUNG
   RUNG wire#w1
      Move(in := "PCComms_TRCV_DB".RCVD_LEN, out1 => "PCComms_Data".RX.BytesReceived)
   END_RUNG
   // the same network as SCL:
   IF "PCComms_TRCV_DB".NDR THEN
       "PCComms_Data".RX.NumberOfSuccesfulReceives := "PCComms_Data".RX.NumberOfSuccesfulReceives + 1;
       "PCComms_Data".RX.BytesReceived := "PCComms_TRCV_DB".RCVD_LEN;
   END_IF;
END_REGION

REGION Network 19: Save the status on an error
   RUNG wire#powerrail
      Contact( "PCComms_TRCV_DB".ERROR )
      Move(in := "PCComms_TRCV_DB".STATUS, out1 => "PCComms_Data".RX.StatusSaved)
   END_RUNG
   // the same network as SCL:
   IF "PCComms_TRCV_DB".ERROR THEN "PCComms_Data".RX.StatusSaved := "PCComms_TRCV_DB".STATUS; END_IF;
END_REGION
END_FUNCTION

FUNCTION "ET_ManageTxBuffer" : Void   // FC742, SCL
{ S7_Optimized_Access := 'TRUE' }
VERSION : 0.0
BEGIN

   //Check if there is a message waiting to be sent and that it is ok to send it
   IF ("ET_TxBuffer".NextAddPoint <> "ET_TxBuffer".LastSendPoint) THEN
       //Incement the send pointer
       "ET_TxBuffer".LastSendPoint := "ET_TxBuffer".LastSendPoint + 1;
       IF ("ET_TxBuffer".LastSendPoint > 10) OR ("ET_TxBuffer".LastSendPoint <= 0) THEN
           "ET_TxBuffer".LastSendPoint := 1;
       END_IF;

       //Copy the data to the transmit area
       "PCComms_Data".EventDataToPC := "ET_TxBuffer".Buffer["ET_TxBuffer".LastSendPoint];

       //Request send is done
       "ET_TxBuffer".SendEvtDataToPCReq := true;
   END_IF;
END_FUNCTION